// TIA Portal V20 export
TYPE "UDT_Service_StringConfigAccessPara"
   STRUCT
      OSLevel : Byte;
      ApplyExt : Bool;
      ApplyOp : Bool;
      Sync : Bool;
      StateOffOp : Bool;
      StateOpOp : Bool;
      StateAutOp : Bool;
      SrcIntOp : Bool;
      SrcExtOp : Bool;
      VExt : String[40];
      VOp : String[40];
   END_STRUCT;
END_TYPE
